PROGRAM MAIN
VAR
END_VAR

FB_GamePlay();

END_PROGRAM

(* stored: Version 1.1.0.1, ProductVersion 3.1.4024.10
   POU MAIN: Id {9defeac3-30d1-4d7a-b475-14fa2c84b25c}, SpecialFunc None *)
